TYPE ST_Tank :
STRUCT
	nId : INT;
	fTemperature : REAL;
	fLevel : REAL;
	bAlarm : BOOL;
	eState : E_TankState;
END_STRUCT
END_TYPE

(* stored: Version 1.1.0.1, ProductVersion 3.1.4024.16
   DUT ST_Tank: Id {eaf29961-2766-4d73-8c06-afacd9f50b96} *)
